(* CoDeSys 2.3.9.37 project: Cap8_1_Res.pro *)
(* Libraries: Standard.lib 4.10.05 12:14:46 *)

(* Global variable list: Global_Variables *)
VAR_GLOBAL
   (* Entradas *)
	Interruptor: BOOL;
   (* Salidas *)
      Luz: BOOL;
END_VAR

(* POU PLC_PRG, LD *)
PROGRAM PLC_PRG
VAR
	MiInter : Intermitente;
END_VAR
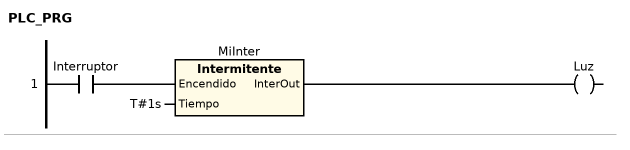
_LD_ (* Ladder Diagram *)
NETWORK 1
	[Interruptor] - MiInter:Intermitente(Encendido: *, Tiempo: T#1s) --- (Luz)
_END_LD_
(* the same logic as Structured Text *)
(* Network 1 *)
MiInter(Encendido := Interruptor, Tiempo := T#1s);
Luz := MiInter.InterOut;
END_PROGRAM

(* POU Intermitente, LD *)
FUNCTION_BLOCK Intermitente
VAR_INPUT
	Encendido : BOOL;
	Tiempo : TIME;
END_VAR
VAR_OUTPUT
	InterOut:BOOL;
END_VAR
VAR
    Tempo: TON;
	Pulso: BOOL;
END_VAR
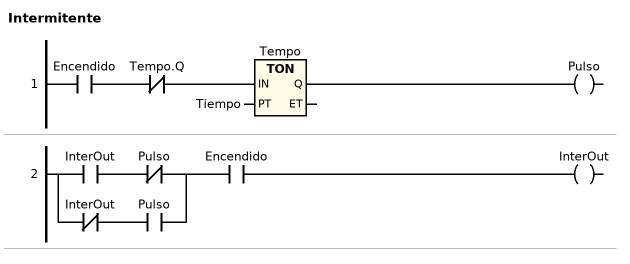
_LD_ (* Ladder Diagram *)
NETWORK 1
	[Encendido] - [/Tempo.Q] - Tempo:TON(IN: *, PT: Tiempo) --- (Pulso)
NETWORK 2
	{ [InterOut] - [/Pulso] | [/InterOut] - [Pulso] } - [Encendido] --- (InterOut)
_END_LD_
(* the same logic as Structured Text *)
(* Network 1 *)
Tempo(IN := Encendido AND NOT Tempo.Q, PT := Tiempo);
Pulso := Tempo.Q;
(* Network 2 *)
InterOut := (InterOut AND NOT Pulso OR NOT InterOut AND Pulso) AND Encendido;
END_FUNCTION_BLOCK

(* Visualisation Visu
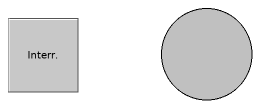
button at (62,99)-(132,173): text "Interr."; toggles Interruptor
ellipse at (215,89)-(306,181): alarm colour if Luz
*)
